// TIA Portal V20 export
DATA_BLOCK "DB_Parameters"   // DB109
// stored: InstanceOfName FB_Parameters, InstanceOfType FB
"FB_Parameters"
   // VAR
   //    Shuttle1Enable : "UDT_BoolEnable";
   //    Shuttle2Enable : Bool;
   // END_VAR
   // VAR RETAIN
   //    GazPressureManual : Real;
   // END_VAR
   // VAR
   //    CoolingVentilatorSetpoint : Real;
   //    TemperatureCoolingSetpoint : Real;
   //    BlowingSetpoint : Real;
   //    sPresenceShuttle1UndrilledPart : "FB_HMI_PLC_Pos";
   //    sPresenceShuttle1UndrilledBw { S7_SetPoint := 'True'} : "FB_HMI_PLC_Pos";
   //    sPresenceShuttle1DrilledPart { S7_SetPoint := 'True'} : "FB_HMI_PLC_Pos";
   //    sPresenceShuttle1DrilledBw { S7_SetPoint := 'True'} : "FB_HMI_PLC_Pos";
   //    sPresenceShuttle2UndrilledPart : "FB_HMI_PLC_Pos";
   //    sPresenceShuttle2UndrilledBw { S7_SetPoint := 'True'} : "FB_HMI_PLC_Pos";
   //    sPresenceShuttle2DrilledPart { S7_SetPoint := 'True'} : "FB_HMI_PLC_Pos";
   //    sPresenceShuttle2DrilledBw { S7_SetPoint := 'True'} : "FB_HMI_PLC_Pos";
   //    sPresenceGripperUndrilledPart : "FB_HMI_PLC_Pos";
   //    sPresenceGripperUndrilledBw { S7_SetPoint := 'True'} : "FB_HMI_PLC_Pos";
   //    sPresenceGripperDrilledPart { S7_SetPoint := 'True'} : "FB_HMI_PLC_Pos";
   //    sPresenceGripperDrilledBw { S7_SetPoint := 'True'} : "FB_HMI_PLC_Pos";
   //    sPresenceFixtureUndrilledPart : "FB_HMI_PLC_Pos";
   //    sPresenceFixtureUndrilledBw { S7_SetPoint := 'True'} : "FB_HMI_PLC_Pos";
   //    sPresenceFixtureDrilledPart { S7_SetPoint := 'True'} : "FB_HMI_PLC_Pos";
   //    sPresenceFixtureDrilledBw { S7_SetPoint := 'True'} : "FB_HMI_PLC_Pos";
   //    sHmiChangeEnable { S7_SetPoint := 'True'} : Bool;
   // END_VAR
BEGIN
END_DATA_BLOCK
